(*
Generates uniformly distributed white noise.

The output is a random value in the range [-:attr:`Amplitude`, +:attr:`Amplitude`]
on every cycle. Useful for testing controller robustness against measurement noise
and disturbances.

.. note::
   The block is ``FINAL`` and must be instantiated, not extended.
   Use ``FB_init`` to set :attr:`Amplitude` at declaration time.
*)
{attribute 'enable_dynamic_creation'}
{attribute 'no_explicit_call' := 'direct call for this function block is not allowed'}
FUNCTION_BLOCK FINAL FB_WhiteNoise EXTENDS FB_SoComponent
IMPLEMENTS FsCommon.I_Runnable
VAR
	_fAmplitude : LREAL; // Maximum absolute output value.
	_fbRng      : FsCommon.FB_RandomNumberGenerator(0); // Internal random number generator.
END_VAR

(*
Gets or sets the amplitude.

The output is uniformly distributed in [-:attr:`Amplitude`, +:attr:`Amplitude`].
A value of 0 holds the output at zero.
*)
PROPERTY Amplitude : LREAL
GET
END_GET
SET
END_SET
END_PROPERTY

METHOD FB_init : BOOL
VAR_INPUT
	bInitRetains : BOOL;  // if TRUE, the retain variables are initialized (warm start / cold start)
	bInCopyCode  : BOOL;  // if TRUE, the instance afterwards gets moved into the copy code (online change)
	fAmplitude   : LREAL; // Maximum absolute output value.
END_VAR
THIS^._fAmplitude := fAmplitude;
END_METHOD

(* Generates the next white noise sample. *)
METHOD Run
VAR_INPUT
END_VAR
THIS^._fOutput := THIS^._fbRng.NextRangedReal(-THIS^._fAmplitude, THIS^._fAmplitude);
END_METHOD

END_FUNCTION_BLOCK

(* stored: Version 1.1.0.1, ProductVersion 3.1.4024.15
   POU FB_WhiteNoise: Id {174d05a6-f244-087d-2ccc-556be2d7466a}, SpecialFunc None
   Property Amplitude: Id {3b120afb-54f2-0b8c-3699-23ef96e57677}
   Get Get: Id {6b35f454-e3a0-04f1-384f-67fc312c835b}
   Set Set: Id {d36c37b4-6a98-06cf-2533-086a8563d362}
   Method FB_init: Id {c02211b8-7557-063c-1ade-7aa48f3e5831}
   Method Run: Id {d26fe23f-0fc4-035c-211f-3101fe5fd07d} *)
